% RSLogix 500 project Project 9.RSS, saved by version 8.30.00.16 %
PROJECT "UNTITLED"    % processor: Bul.1763 MicroLogix 1100 Series B %

PROGRAM FILES
  LAD 2   8 rungs

DATA FILES
  O0 OUTPUT  4 elements
  I1 INPUT  6 elements
  S2 STATUS  66 elements
  B3 BINARY  1 elements
  T4 TIMER  1 elements
  C5 COUNTER  1 elements
  R6 CONTROL  1 elements
  N7 INTEGER  4 elements
  F8 FLOAT  1 elements
  ST9 STRING  11 elements

LADDER 2
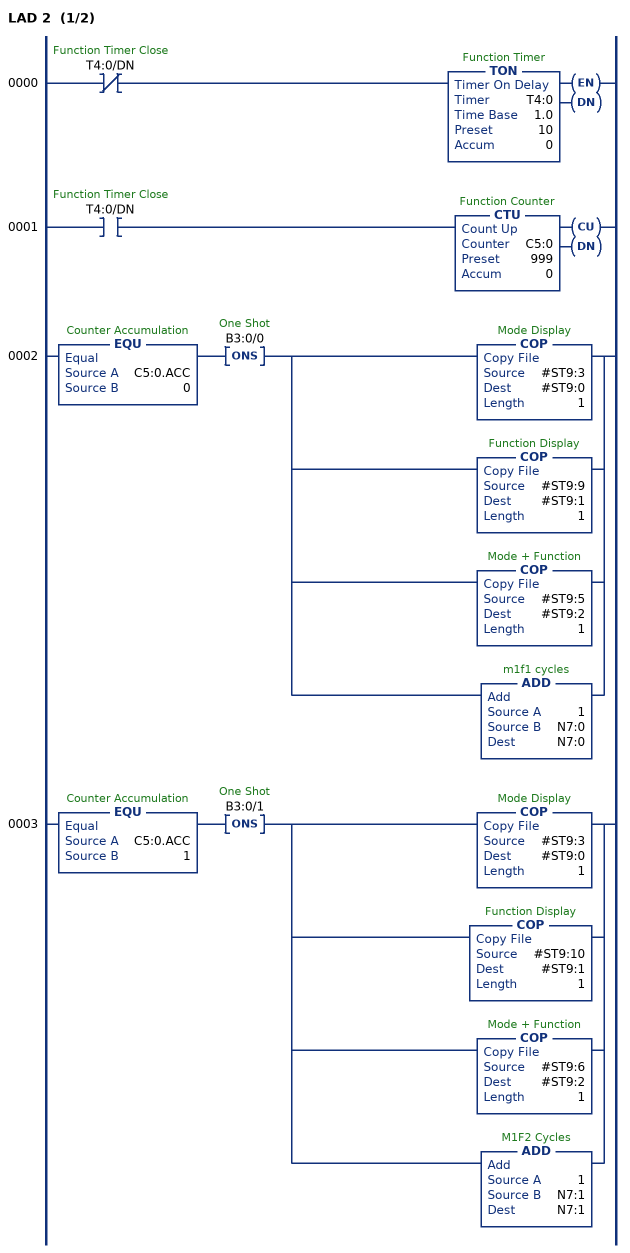
% Rung: 0 %
SOR XIO T4:0/DN TON T4:0 1.0 10 0 EOR
%   T4:0/DN  "Function Timer Close" %
%   T4:0  "Function Timer" %
% Rung: 1 %
SOR XIC T4:0/DN CTU C5:0 999 0 EOR
%   T4:0/DN  "Function Timer Close" %
%   C5:0  "Function Counter" %
% Rung: 2 %
SOR EQU C5:0.ACC 0 ONS B3:0/0 BST COP #ST9:3 #ST9:0 1 NXB COP #ST9:9 #ST9:1 1 NXB COP #ST9:5 #ST9:2 1 NXB ADD 1 N7:0 N7:0 BND EOR
%   C5:0.ACC  "Counter Accumulation" %
%   B3:0/0  "One Shot" %
%   ST9:3  "Mode 1" %
%   ST9:0  "Mode Display" %
%   ST9:9  "Function 1" %
%   ST9:1  "Function Display" %
%   ST9:5  "M1F1" %
%   ST9:2  "Mode + Function" %
%   N7:0  "m1f1 cycles" %
% Rung: 3 %
SOR EQU C5:0.ACC 1 ONS B3:0/1 BST COP #ST9:3 #ST9:0 1 NXB COP #ST9:10 #ST9:1 1 NXB COP #ST9:6 #ST9:2 1 NXB ADD 1 N7:1 N7:1 BND EOR
%   C5:0.ACC  "Counter Accumulation" %
%   B3:0/1  "One Shot" %
%   ST9:3  "Mode 1" %
%   ST9:0  "Mode Display" %
%   ST9:10  "Function 2" %
%   ST9:1  "Function Display" %
%   ST9:6  "M1F2" %
%   ST9:2  "Mode + Function" %
%   N7:1  "M1F2 Cycles" %

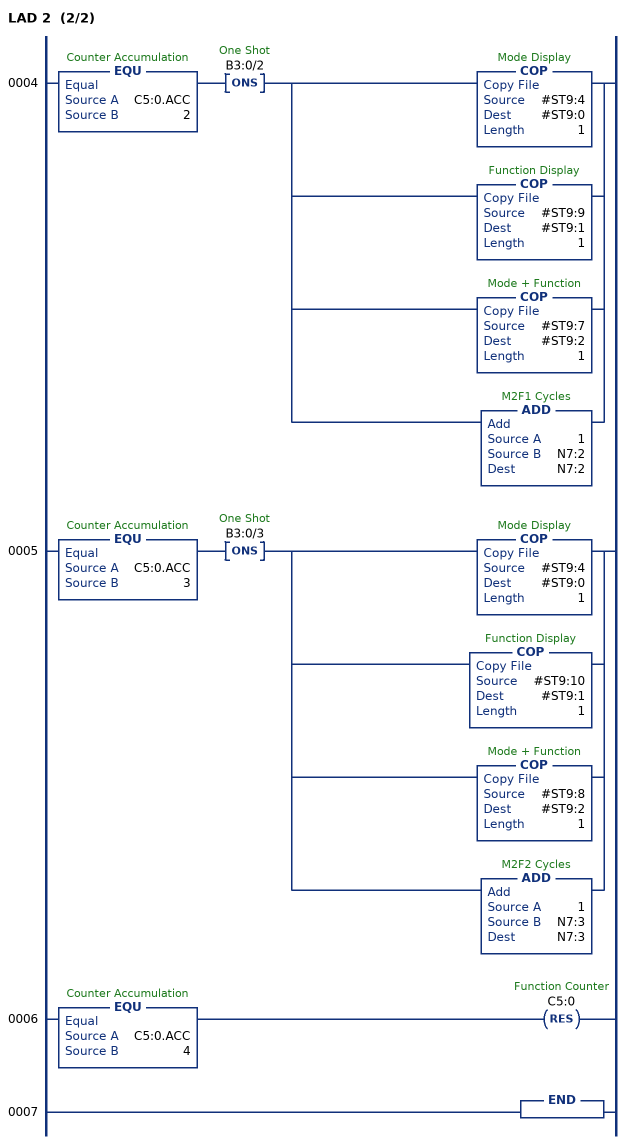
% Rung: 4 %
SOR EQU C5:0.ACC 2 ONS B3:0/2 BST COP #ST9:4 #ST9:0 1 NXB COP #ST9:9 #ST9:1 1 NXB COP #ST9:7 #ST9:2 1 NXB ADD 1 N7:2 N7:2 BND EOR
%   C5:0.ACC  "Counter Accumulation" %
%   B3:0/2  "One Shot" %
%   ST9:4  "Mode 2" %
%   ST9:0  "Mode Display" %
%   ST9:9  "Function 1" %
%   ST9:1  "Function Display" %
%   ST9:7  "M2F1" %
%   ST9:2  "Mode + Function" %
%   N7:2  "M2F1 Cycles" %
% Rung: 5 %
SOR EQU C5:0.ACC 3 ONS B3:0/3 BST COP #ST9:4 #ST9:0 1 NXB COP #ST9:10 #ST9:1 1 NXB COP #ST9:8 #ST9:2 1 NXB ADD 1 N7:3 N7:3 BND EOR
%   C5:0.ACC  "Counter Accumulation" %
%   B3:0/3  "One Shot" %
%   ST9:4  "Mode 2" %
%   ST9:0  "Mode Display" %
%   ST9:10  "Function 2" %
%   ST9:1  "Function Display" %
%   ST9:8  "M2F2" %
%   ST9:2  "Mode + Function" %
%   N7:3  "M2F2 Cycles" %
% Rung: 6 %
SOR EQU C5:0.ACC 4 RES C5:0 EOR
%   C5:0.ACC  "Counter Accumulation" %
%   C5:0  "Function Counter" %
% Rung: 7 %
SOR END EOR

DATA TABLE (non-zero values as saved)
DATA T4
% .PRE .ACC %
% T4:0 % 10 0
DATA C5
% .PRE .ACC %
% C5:0 % 999 0
DATA ST9
% ST9:3 % "Mode-1"
% ST9:4 % "Mode-2"
% ST9:5 % "M1F1"
% ST9:6 % "M1F2"
% ST9:7 % "M2F1"
% ST9:8 % "M2F2"
% ST9:9 % "F1"
% ST9:10 % "F2"
